TYPE ST_OvercurrentProtection_Events :
STRUCT
	Input	:ARRAY [1..2] OF ARRAY [1..4] OF FB_Overcurrentdetect(); //FB_UpperLimitAndTimeExceeded();
	Output	:ARRAY [1..3] OF ARRAY [1..4] OF FB_Overcurrentdetect();
END_STRUCT
END_TYPE

(* stored: Version 1.1.0.1, ProductVersion 3.1.4026.18
   DUT ST_OvercurrentProtection_Events: Id {a88aee90-2a5c-472d-a9cf-ee5c1a849c99} *)
